(*

.. <legal notes>

legal notes
=================
| SPDX-FileCopyrightText: © 2026 Oleksandr Tiutyk <trofimich@gmail.com>
| SPDX-License-Identifier: LGPL-3.0-only
| For details check: LGPL-3.0-only_

.. _LGPL-3.0-only: https://www.gnu.org/licenses/lgpl-3.0.en.html

.. </legal notes>

*)

INTERFACE IDevice EXTENDS IAutomationComponent

METHOD Initialize : BOOL
END_METHOD

{attribute 'monitoring' := 'call'}
PROPERTY Parent : IAutomationComponent
GET
END_GET
END_PROPERTY

METHOD ABSTRACT Recover
END_METHOD

END_INTERFACE

(* stored: Version 1.1.0.1
   Itf IDevice: Id {9736df80-aba4-4bb1-a085-478863d519b5}
   Method Initialize: Id {c1b642e1-c838-4d11-be0f-d347cee28d0c}
   Property Parent: Id {2297a1f3-aeb4-4b46-9b02-c8e14801ec7a}
   Get Get: Id {e145fc3f-3a76-4e5b-b248-c246c2e58910}
   Method Recover: Id {213e8bf7-9733-43de-b1a2-ec38a779dbf6} *)
